TYPE U_Fanuc_Out :
UNION
	aFanuc_Out		AT %Q*	:ARRAY [1..16] OF BYTE;
	stFanucOut				:ST_Fanuc_Out;
END_UNION
END_TYPE

(* stored: Version 1.1.0.1, ProductVersion 3.1.4024.11
   DUT U_Fanuc_Out: Id {29d70634-92fe-4c86-aa57-93adc0705f55} *)
